FUNCTION_BLOCK PlaceServices (* Composite Function Block Type *)
  (* Standard: 61499-2 *)
  (* Version 0.0, 11/3/2020, prana, nxtControl GmbH, template *)
  PACKAGE Main;
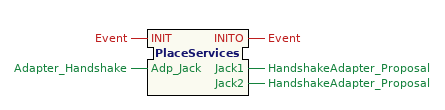
  EVENT_INPUT
    INIT; (* Initialization Request *)
  END_EVENT
  EVENT_OUTPUT
    INITO; (* Initialization Confirm *)
  END_EVENT
  SOCKETS
    Adp_Jack : Adapter_Handshake;
  END_SOCKETS
  PLUGS
    Jack1 : HandshakeAdapter_Proposal;
    Jack2 : HandshakeAdapter_Proposal;
  END_PLUGS
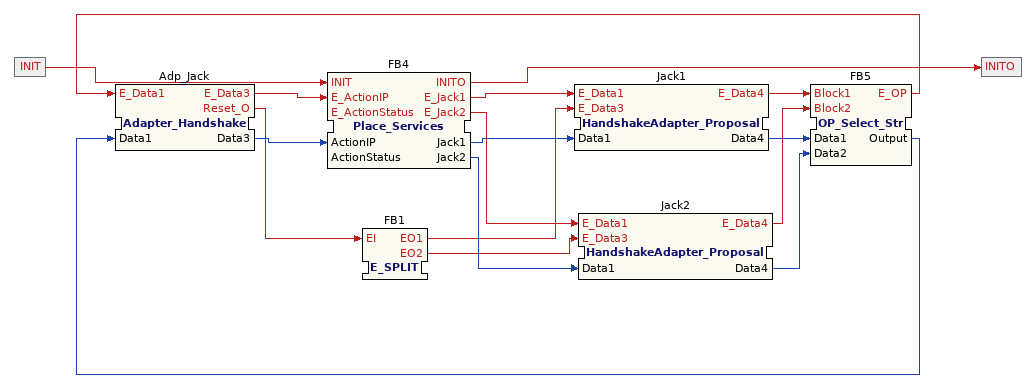
  FBS
    FB4 : Place_Services;
    FB5 : OP_Select_Str;
    FB1 : E_SPLIT;
  END_FBS
  EVENT_CONNECTIONS
    FB4.E_Jack1 TO Jack1.E_Data1;
    FB4.E_Jack2 TO Jack2.E_Data1;
    Jack1.E_Data4 TO FB5.Block1;
    Jack2.E_Data4 TO FB5.Block2;
    Adp_Jack.E_Data3 TO FB4.E_ActionIP;
    INIT TO FB4.INIT;
    FB4.INITO TO INITO;
    Adp_Jack.Reset_O TO FB1.EI;
    FB1.EO1 TO Jack1.E_Data3;
    FB1.EO2 TO Jack2.E_Data3;
    FB5.E_OP TO Adp_Jack.E_Data1;
  END_CONNECTIONS
  DATA_CONNECTIONS
    FB4.Jack1 TO Jack1.Data1;
    FB4.Jack2 TO Jack2.Data1;
    Jack1.Data4 TO FB5.Data1;
    Jack2.Data4 TO FB5.Data2;
    Adp_Jack.Data3 TO FB4.ActionIP;
    FB5.Output TO Adp_Jack.Data1;
  END_CONNECTIONS
END_FUNCTION_BLOCK
